// TwinCAT 3 PLC project CarlPlc
// ProgramVersion: 3.1.4022.1
// libraries:
//   Tc2_ModbusRTU, * (Beckhoff Automation GmbH)
//   Tc2_Standard, * (Beckhoff Automation GmbH)
//   Tc2_System, * (Beckhoff Automation GmbH)
//   Tc2_Utilities, * (Beckhoff Automation GmbH)
//   Tc3_Module, * (Beckhoff Automation GmbH)
//   BASIC,3.3.3.0,OSCAT
// project tree:
//   Common/ DetectEvent.TcPOU (not stored), GVL_Common.TcGVL (not stored), TasterEventStates.TcDUT, TasterEventType.TcDUT (not stored), LinearCalibration.TcDUT (not stored)
//   FlowRateSensor/ GVL_FlowControl.TcGVL (not stored), PRG_UpdateFlowRateSensor.TcPOU
//   GasAnalysis/ GVL_GasAnalysis.TcGVL, PRG_GasAnalysis.TcPOU (not stored)
//   GasSupply/ GVL_GasSupply.TcGVL (not stored), PRG_UpdateGasSupply.TcPOU (not stored)
//   MotorControl/ GVL_MotorControl.TcGVL, PRG_UpdateMotor.TcPOU (not stored)
//   pHOrpControl/ EN_ModbusReadTarget.TcDUT (not stored), GVL_PhOrpControl.TcGVL (not stored), PRG_ReadModbusSensorData.TcPOU, PRG_UpdatePhControl.TcPOU (not stored)
//   / PlcTask.TcTTO (not stored)
//   MAIN/ MAIN.TcPOU (not stored)
//   ReactorPressureControl/ GVL_ReactorPressureControl.TcGVL (not stored), PRG_UpdatePressureSensor.TcPOU (not stored)
//   RoomTempRh/ GVL_TempRHSensor.TcGVL, PRG_UpdateRoomTempRh.TcPOU (not stored)
//   TemperatureControl/ EN_TempControlMode.TcDUT (not stored), FB_TON.TcPOU (not stored), GVL_TemperatureControl.TcGVL, FUN_ComputeMovingSetPoint.TcPOU, PRG_UpdateTemperatureControl.TcPOU
//   TemperatureControl/PID/ CLK_PRG.TcPOU, FB_PWM.TcPOU (not stored), FT_DERIV.TcPOU (not stored), FT_PIDWL.TcPOU, FT_PIWL.TcPOU, PWM_DC.TcPOU (not stored), TP_X.TcPOU (not stored), T_PLC_MS.TcPOU (not stored), T_PLC_US.TcPOU
// real-time tasks:
//   TASK PlcTask: cycle T#10ms, priority 20, ADS port 350
// I/O:
//   DEVICE Device 1 (EtherCAT), AmsNetId 5.54.16.198.2.1
//     Term 1 (EK1200) [EK1200-5000 EtherCAT Power supply (2A E-Bus)]
//       Term 2 (EL3014) Motor Speed In [EL3014 4Ch. Ana. Input 0-20mA DIFF]
//       Term 3 (EL4004) Motor Speed Out [EL4004 4Ch. Ana. Output 0-10V, 12bit]
//       Term 4 (EL2004) DO Heating Cooling [EL2004 4Ch. Dig. Output 24V, 0.5A]
//       Term 5 (EL2004) DO Gassing Valves [EL2004 4Ch. Dig. Output 24V, 0.5A]
//       Term 6 (EL2004) DO Motor Control Out [EL2004 4Ch. Dig. Output 24V, 0.5A]
//       Term 7 (EL6021) PhModbus [EL6021 Interface (RS422/485)]
//       Term 8 (EL6021) OrpModbus [EL6021 Interface (RS422/485)]
//       Term 21 (EL1004) DI Gas Analysis [EL1004 4Ch. Dig. Input 24V, 3ms]
//       Term 18 (EL3052) AI Pressure Flow [EL3052 2Ch. Ana. Input 4-20mA]
//       Term 24 (EL3052) AI Heating Cooling [EL3052 2Ch. Ana. Input 4-20mA]
//       Term 10 (EL9184) [EL9184 Potential Connection, 8 x 24V, 8 x Ground]
//       Term 26 (EL3044) [EL3044 4Ch. Ana. Input 0-20mA]
//       Term 9 (EL9011) [EL9011 End Terminal]
// variable links:
//   CarlPlc/CarlPlc Instance <-> Device 1 (EtherCAT)/Term 1 (EK1200)/Term 18 (EL3052) AI Pressure Flow
//     PlcTask Inputs/GVL_FlowControl.flowRateRawCounts <-> FlowRateSensor/FlowRateRaw
//     PlcTask Inputs/GVL_ReactorPressureControl.pressureRawCounts <-> PressureSensor/PressureSensorRaw
//   CarlPlc/CarlPlc Instance <-> Device 1 (EtherCAT)/Term 1 (EK1200)/Term 2 (EL3014) Motor Speed In
//     PlcTask Inputs/GVL_MotorControl.motorActualSpeed <-> AI Motor RPM/Value
//     PlcTask Inputs/GVL_TempRHSensor.roomRhRaw <-> AI Room RH/Value
//     PlcTask Inputs/GVL_TempRHSensor.roomTempRaw <-> AI Room Temp/Value
//   CarlPlc/CarlPlc Instance <-> Device 1 (EtherCAT)/Term 1 (EK1200)/Term 21 (EL1004) DI Gas Analysis
//     PlcTask Inputs/GVL_GasAnalysis.ch4FlowSensor <-> Flow Sensor CH4/Input
//     PlcTask Inputs/GVL_GasAnalysis.o2FlowSensor <-> Flow Sensor O2/Input
//   CarlPlc/CarlPlc Instance <-> Device 1 (EtherCAT)/Term 1 (EK1200)/Term 24 (EL3052) AI Heating Cooling
//     PlcTask Inputs/GVL_TemperatureControl.jacketTempRaw <-> AI Jacket Temp/Value
//   CarlPlc/CarlPlc Instance <-> Device 1 (EtherCAT)/Term 1 (EK1200)/Term 26 (EL3044)
//     PlcTask Inputs/GVL_GasAnalysis.ch4SensorRaw <-> AI CH4/Value
//     PlcTask Inputs/GVL_GasAnalysis.o2SensorRaw <-> AI O2/Value
//     PlcTask Inputs/GVL_GasSupply.gasSupplyPressureRaw <-> AI Gas Supply Pressure/Value
//   CarlPlc/CarlPlc Instance <-> Device 1 (EtherCAT)/Term 1 (EK1200)/Term 3 (EL4004) Motor Speed Out
//     PlcTask Outputs/GVL_MotorControl.motorTargetSpeed <-> MotorTargetSpeed/MotorTargetSpeed
//     PlcTask Outputs/GVL_PhOrpControl.acidPumpSpeedCount <-> AcidPumpSpeedCount/acidPumpSpeedCount
//   CarlPlc/CarlPlc Instance <-> Device 1 (EtherCAT)/Term 1 (EK1200)/Term 4 (EL2004) DO Heating Cooling
//     PlcTask Outputs/GVL_TemperatureControl.coldValve <-> ColdValve/Output
//     PlcTask Outputs/GVL_TemperatureControl.hotValve <-> HotValve/Output
//     PlcTask Outputs/GVL_TemperatureControl.pumpOn <-> PumpOn/Output
//     PlcTask Outputs/GVL_TemperatureControl.steriValve <-> SteriValve/Output
//   CarlPlc/CarlPlc Instance <-> Device 1 (EtherCAT)/Term 1 (EK1200)/Term 5 (EL2004) DO Gassing Valves
//     PlcTask Outputs/GVL_GasSupply.gasSupplyValve <-> GasSupplyValve/Output
//     PlcTask Outputs/GVL_ReactorPressureControl.reactorPressureInletValve <-> reactorPressureInlet/ReactorPressureInlet
//     PlcTask Outputs/GVL_ReactorPressureControl.reactorPressureOutletValve <-> reactorPressureOutlet/Output
//   CarlPlc/CarlPlc Instance <-> Device 1 (EtherCAT)/Term 1 (EK1200)/Term 6 (EL2004) DO Motor Control Out
//     PlcTask Outputs/GVL_MotorControl.motorReset <-> motorReset/Output
//     PlcTask Outputs/GVL_MotorControl.motorStart <-> motorStart/Output
//   CarlPlc/CarlPlc Instance <-> Device 1 (EtherCAT)/Term 1 (EK1200)/Term 7 (EL6021) PhModbus
//     PlcTask Inputs/GVL_Common.PhModbus.InData/D[{0..21}] <-> COM TxPDO-Map Inputs/Data In {0..21}  (22 links)
//     PlcTask Inputs/GVL_Common.PhModbus.InData/Status <-> COM TxPDO-Map Inputs/Status
//     PlcTask Outputs/GVL_Common.PhModbus.OutData/Ctrl <-> COM RxPDO-Map Outputs/Ctrl
//     PlcTask Outputs/GVL_Common.PhModbus.OutData/D[{0..21}] <-> COM RxPDO-Map Outputs/Data Out {0..21}  (22 links)
//   CarlPlc/CarlPlc Instance <-> Device 1 (EtherCAT)/Term 1 (EK1200)/Term 8 (EL6021) OrpModbus
//     PlcTask Inputs/GVL_Common.OrpModbus.InData/D[{0..21}] <-> COM TxPDO-Map Inputs/Data In {0..21}  (22 links)
//     PlcTask Inputs/GVL_Common.OrpModbus.InData/Status <-> COM TxPDO-Map Inputs/Status
//     PlcTask Outputs/GVL_Common.OrpModbus.OutData/Ctrl <-> COM RxPDO-Map Outputs/Ctrl
//     PlcTask Outputs/GVL_Common.OrpModbus.OutData/D[{0..21}] <-> COM RxPDO-Map Outputs/Data Out {0..21}  (22 links)

// ---- Common/TasterEventStates.TcDUT
TYPE TasterEventStates : (TASTEVTST_Init := 0,
						TASTEVTST_FirstPosEdge,
						TASTEVTST_FirstNegEdge,
						TASTEVTST_FirstLongClick);
END_TYPE

// ---- GasAnalysis/GVL_GasAnalysis.TcGVL
VAR_GLOBAL
	ch4FlowSensor			AT %I*	: BOOL;
	o2FlowSensor			AT %I*	: BOOL;
	
	ch4SensorRaw			AT %I*	: INT;
	o2SensorRaw 			AT %I*	: INT;
	
	ch4ValuemA				: REAL := 0.0;
	o2ValuemA				: REAL := 0.0;
	
	ch4ValuePercent			: REAL := 0.0;
	o2ValuePercent			: REAL := 0.0;
	
	ch4CalibrationToPercent : LinearCalibration := (scaleFactor := 8.3415719228868017795353435491844E-5, offset := 0.3);
	ch4CalibrationToMa		: LinearCalibration := (scaleFactor := 20.0/32768.0, offset := 0.0);
	o2CalibrationToPercent	: LinearCalibration := (scaleFactor := 8.3415719228868017795353435491844E-5, offset := 0.3);
	o2CalibrationToMa		: LinearCalibration := (scaleFactor := 20.0/32768.0, offset := 0.0);
	
	(* Sensor Status *)
	ch4SensorStatus			: INT  := 0; 	(* 0: FAULT (1mA output), 1: BEAMBLOCK(2mA output), 2: STARTUP (3mA output), 3: Running (4 > 20 mA output) *)

	o2SensorFault			: BOOL := FALSE;
	
	gasAnalysisControlStartStop : BOOL := FALSE;
	gasAnalysisControlManual	: BOOL := FALSE;
	
	gasAnalysisValveAutomatic	: BOOL := FALSE;
	gasAnalysisValveManual 		: BOOL := FALSE;	

END_VAR


VAR_GLOBAL PERSISTENT
	ch4ValuePercentSet			: REAL := 0.0;
	gasAnalysisControlRunning 	: BOOL;
END_VAR

// ---- MotorControl/GVL_MotorControl.TcGVL
VAR_GLOBAL
	(* agitation motor *)	
	motorActualSpeed 	AT %I*	: INT;
	motorTargetSpeed 	AT %Q*	: INT;
	
	motorRpm					: INT; 
	
	(* motor target speed setting --> see retains *)
	motorStart			AT %Q*	: BOOL := FALSE;
	motorReset			AT %Q*	: BOOL := FALSE;
	
	motorStartButton			: BOOL := FALSE;
	motorStopButton				: BOOL := FALSE;
	motorResetButton			: BOOL := FALSE;

	(* motorIsRunning				: BOOL := FALSE; *)
END_VAR

VAR_GLOBAL PERSISTENT
	motorRunning				: BOOL;
	currentMotorSpeedSetting	: INT;
END_VAR

// ---- RoomTempRh/GVL_TempRHSensor.TcGVL
VAR_GLOBAL
	roomTempRaw			AT %I*	: INT;
	roomRhRaw 			AT %I*	: INT;	
	
	roomTemp			: REAL;
	roomRh				: REAL;
END_VAR

// ---- TemperatureControl/GVL_TemperatureControl.TcGVL
VAR_GLOBAL


	tPhCurrent					: REAL := 0.0;
	tPhLastReadingValid			: BOOL := FALSE;
	tOrpCurrent					: REAL := 0.0;
	tOrpLastReadingValid		: BOOL := FALSE;


	(* temperature control *)
	pumpOn				AT %Q* 	: BOOL := FALSE;
	coldValve			AT %Q* 	: BOOL := FALSE;
	hotValve			AT %Q* 	: BOOL := FALSE;
	steriValve			AT %Q*	: BOOL := FALSE; 
	
	jacketTempRaw		AT %I*	: INT;
	jacketTempC					: REAL := 0.0;
	jacketTempK					: REAL := 0.0;
	
	
	tempControlStop				: BOOL := FALSE;
	tempControlStart			: BOOL := FALSE;
	hotValveButton				: BOOL := FALSE;
	coldValveButton				: BOOL := FALSE;
	
	pumpIsRunning				: BOOL := FALSE;
	tempControlRunning			: BOOL := FALSE;
	tempSafetyEnabled			: BOOL := FALSE;
	
	steriStart					: BOOL := FALSE;
	steriStop					: BOOL := FALSE;
	steriRunning				: BOOL := FALSE;

	
	currentMeanTemp				: REAL := 0;
	currentTempValid			: BOOL := FALSE;
	(* target temp -> see retains *) 
	
	tempIsBelowSteriTemp		: BOOL := TRUE;
	(* target steri temp --> see retains *)	

	
END_VAR

VAR_GLOBAL PERSISTENT
	targetControlTemp			: REAL;
	targetSteriTemp				: REAL;
	targetSteriTimeMinutes		: INT;
	remainingSteriTimeMinutes	: REAL;
	
	
	remainingSteriTimeInMs		: DINT; (* 30 min in ms *)
	
	countTempSpikes				: INT;
	countValveMaxTimeExceeded	: INT;

	pidResetCounter				: INT;
END_VAR

VAR_GLOBAL CONSTANT
	CYCLE_TIME_IN_MS		: TIME := T#10ms;
END_VAR

// ---- pHOrpControl/PRG_ReadModbusSensorData.TcPOU
PROGRAM PRG_ReadModbusSensorData
VAR
	
	CurrentReadTarget			: EN_ModbusReadTarget := EN_ModbusReadTarget.READ_TARGET_PH;
	
	ProcessValueRegister		: WORD := 2089;
	TemperatureRegister			: WORD := 2409;
	PhSensorUnitId				: BYTE := 1;
	OrpSensorUnitId				: BYTE := 2;
	RegQuantityToRead			: WORD :=10;
	
	currentUnitId				: BYTE := PhSensorUnitId;
	currentModbusRegister		: WORD := ProcessValueRegister;

	ModbusBusy					: BOOL := FALSE;

	(* diagnostics *)	
	LastModbusError				: ST_ModbusErrorDiagnostics;
	LastErrorstate				: INT;
	CurrentState				: INT;
	CounterError				: INT := 0;
	CounterSuccess				: INT := 0;
	
	firstCall					: BOOL := TRUE;	
	
	scaleFactorPh				: REAL :=   1.219512195; (* 0.980167935 *);  		
	offsetPh					: REAL := 	-1.280487805; (* -0.0216290391086993 *);	


	scaleFactorOrp				: REAL := 0.999321727334388;
	offsetOrp					: REAL := 0.0;			
	
END_VAR

(* looping through pH, pH-T, ORP, ORP-T reading the latest values *)
IF firstCall THEN
	PhModbus.ReadRegs( Execute := FALSE);
	OrpModbus.ReadRegs( Execute := FALSE);
	firstCall := FALSE;
END_IF	

CASE  CurrentReadTarget OF 
	EN_ModbusReadTarget.READ_TARGET_PH:
		PhModbus.Readregs (UnitID 		:= PhSensorUnitId ,
   							Quantity   	:= RegQuantityToRead,
   							MBAddr    	:= ProcessValueRegister,
   							cbLength    := RegQuantityToRead*2,
   							pMemoryAddr := ADR(PhValueArrayIn),   
   							Execute    	:= TRUE,
   							Timeout    	:= T#300MS,
							Busy 		=> ModbusBusy	
						  );
		
		IF NOT ModbusBusy THEN
			PhModbus.ReadRegs(Execute:= FALSE);
			CurrentReadTarget := EN_ModbusReadTarget.READ_TARGET_PH_T;
	
			IF PhModbus.Error THEN
				LastModbusError 	:= PhModbus.ErrorDiagnostics;
				LastErrorstate 		:= CurrentState;
				CounterError 		:= CounterError + 1;
				phLastReadingValid 	:= FALSE;
			ELSE
				CounterSuccess 		:= CounterSuccess + 1;
				phLastReadingValid 	:= TRUE;
				phCurrent			:= PhValueArrayIn[1]*scaleFactorPh + offsetPh;
			END_IF
		END_IF
		
	EN_ModbusReadTarget.READ_TARGET_PH_T:
		PhModbus.Readregs (UnitID 		:= PhSensorUnitId ,
   							Quantity   	:= RegQuantityToRead,
   							MBAddr    	:= TemperatureRegister,
   							cbLength    := RegQuantityToRead*2,
   							pMemoryAddr := ADR(TPhValueArrayIn),   
   							Execute    	:= TRUE,
   							Timeout    	:= T#300MS,
							Busy 		=> ModbusBusy	
						  );
		
		IF NOT ModbusBusy THEN
			PhModbus.ReadRegs(Execute:= FALSE);	
			CurrentReadTarget := EN_ModbusReadTarget.READ_TARGET_ORP;

			IF PhModbus.Error THEN
				LastModbusError 	:= PhModbus.ErrorDiagnostics;
				LastErrorstate 		:= CurrentState;
				CounterError 		:= CounterError + 1;
				tPhLastReadingValid := FALSE;
			ELSE
				CounterSuccess 		:= CounterSuccess + 1;
				tPhLastReadingValid := TRUE;
				tPhCurrent			:= TPhValueArrayIn[1];
			END_IF
		END_IF
	
	EN_ModbusReadTarget.READ_TARGET_ORP:
		OrpModbus.Readregs (UnitID 		:= OrpSensorUnitId ,
   							Quantity   	:= RegQuantityToRead,
   							MBAddr    	:= ProcessValueRegister,
   							cbLength    := RegQuantityToRead*2,
   							pMemoryAddr := ADR(OrpValueArrayIn),   
   							Execute    	:= TRUE,
   							Timeout    	:= T#300MS,
							Busy 		=> ModbusBusy	
						  );
		
		IF NOT ModbusBusy THEN
			OrpModbus.ReadRegs(Execute:= FALSE);	
			CurrentReadTarget := EN_ModbusReadTarget.READ_TARGET_ORP_T;

			IF OrpModbus.Error THEN
				LastModbusError 	:= OrpModbus.ErrorDiagnostics;
				LastErrorstate 		:= CurrentState;
				CounterError 		:= CounterError + 1;
				orpLastReadingValid := FALSE;
			ELSE
				CounterSuccess 		:= CounterSuccess + 1;
				orpLastReadingValid := TRUE;
				orpCurrent			:= OrpValueArrayIn[1]*scaleFactorOrp + offsetOrp;
			END_IF
		END_IF

	EN_ModbusReadTarget.READ_TARGET_ORP_T:

		OrpModbus.Readregs (UnitID 		:= OrpSensorUnitId ,
   							Quantity   	:= RegQuantityToRead,
   							MBAddr    	:= TemperatureRegister,
   							cbLength    := RegQuantityToRead*2,
   							pMemoryAddr := ADR(TOrpValueArrayIn),   
   							Execute    	:= TRUE,
   							Timeout    	:= T#300MS,
							Busy 		=> ModbusBusy	
						  );
		
		IF NOT ModbusBusy THEN
			OrpModbus.ReadRegs(Execute:= FALSE);	
			CurrentReadTarget := EN_ModbusReadTarget.READ_TARGET_PH;

			IF OrpModbus.Error THEN
				LastModbusError := OrpModbus.ErrorDiagnostics;
				LastErrorstate 	:= CurrentState;
				CounterError 	:= CounterError + 1;
				tOrpLastReadingValid := FALSE;
			ELSE
				CounterSuccess 	:= CounterSuccess + 1;
				tOrpLastReadingValid := TRUE;
				tOrpCurrent	:= TOrpValueArrayIn[1];
			END_IF
		END_IF
	
END_CASE
			
IF tPhLastReadingValid AND tOrpLastReadingValid THEN
	currentMeanTemp := (tPhCurrent + tOrpCurrent)/2.0;
	currentTempValid := TRUE;
ELSIF tPhLastReadingValid AND NOT tOrpLastReadingValid THEN
	currentMeanTemp := tPhCurrent;
	currentTempValid := TRUE;
ELSIF NOT tPhLastReadingValid AND tOrpLastReadingValid THEN
	currentMeanTemp := tOrpCurrent;
	currentTempValid := TRUE;
ELSE 
	(* no valid temperature signal !! signal to stop temperature control, if active *)
	currentTempValid := FALSE;
END_IF

END_PROGRAM

// ---- FlowRateSensor/PRG_UpdateFlowRateSensor.TcPOU
PROGRAM PRG_UpdateFlowRateSensor
VAR
	deltaVolume : REAL := 0.0;
END_VAR

IF flowRateRawCounts < 20 THEN
	flowRateLitersPerMinute := 0.0;
ELSE
	flowRateLitersPerMinute := INT_TO_REAL(flowRateRawCounts)*flowRateCalibration.scaleFactor + flowRateCalibration.offset;
END_IF

deltaVolume := flowRateLitersPerMinute*0.01/60.0;
spargeVolume := spargeVolume + deltaVolume;
spargeVolumeCumulative := spargeVolumeCumulative+ deltaVolume;

IF  resetSpargeVolume THEN
	resetSpargeVolume := FALSE;
	spargeVolume := 0.0;
END_IF

IF resetSpargeVolumeCumulative THEN
	resetSpargeVolumeCumulative := FALSE;
	spargeVolumeCumulative := 0.0;
END_IF

END_PROGRAM

// ---- TemperatureControl/PID/CLK_PRG.TcPOU
	FUNCTION_BLOCK CLK_PRG
VAR_INPUT
	PT : TIME := t#10ms;
END_VAR
VAR_OUTPUT
	Q : BOOL;
END_VAR
VAR
	init : BOOL;
	last : TIME;
	tx: TIME;
END_VAR

(*clk_prg uses the internal sps time to generate a clock with programmable period time.
the period time is defined for 10ms .. 65s
the first cycle after start is a clk pulse and then depending on the programmed period time a delay.
every pulse is only valid for one cycle.
the accuracy of clk_prg is depending on the accuracy of the system clock.*)

(* read system time *)
tx := DWORD_TO_TIME(T_PLC_MS());

(* initialize on startup *)
IF NOT init THEN
	init := TRUE;
	last := tx - pt;
END_IF;

(* generate output pulse when next_pulse is reached *)
Q := tx - last >= pt;
IF Q THEN last := tx; END_IF;

END_FUNCTION_BLOCK

// ---- TemperatureControl/PID/FT_PIDWL.TcPOU
FUNCTION_BLOCK FT_PIDWL
VAR_INPUT
	IN : REAL;
	KP : REAL := 1.0;
	TN : REAL := 1.0;
	TV : REAL := 1.0;
	LIM_L : REAL := -1.0E38;
	LIM_H : REAL := 1.0E38;
	RST : BOOL;
END_VAR
VAR_OUTPUT
	Y : REAL;
	LIM : BOOL;
END_VAR
VAR
	piwl : FT_PIWL;
	diff : FT_DERIV;
END_VAR

(*
version 1.3	13. nov. 2009
programmer 	hugo
tested by		tobias

FT_PIDWL is a PID controller with dynamic wind_up reset.
The PID controller works according to the fomula Y = KP *(IN + KI * INTEG(e) + DERIV(e) ).
a rst will reset the integrator to 0
lim_h and Lim_l set the possible output range of the internal integrator.
the output flags lim will signal that the output limits are active.

default values for KP = 1, KI = 1, ILIM_L = -1E37, iLIM_H = +1E38.
*)

(* if rst then *)
IF rst THEN
	piwl(rst := TRUE);
	piwl.RST := FALSE;
ELSE
	(* run PIWL controller first *)
	(* we need to check if TN = 0 and do alternative calls *)
	IF TN = 0.0 THEN
		piwl(in := IN * KP, KP := 1.0, KI := 0.0, LIM_L := LIM_L, LIM_H := LIM_H);
	ELSE
		piwl(in := IN * KP, KP := 1.0, KI := 1.0 / TN, LIM_L := LIM_L, LIM_H := LIM_H);
	END_IF;

	(* run differentiator and add_to_output *)
	diff(IN := IN, K := TV);
	Y := piwl.Y + diff.out;

	(* limit the output *)
	IF Y < LIM_L THEN
		LIM := TRUE;
		Y := LIM_L;
	ELSIF Y > LIM_H THEN
		LIM := TRUE;
		Y := LIM_H;
	ELSE
		LIM := FALSE;
	END_IF;
END_IF;



(* revision history
hm 13. jun. 2008 	rev 1.0
	original version

hm	25. jan 2008	rev 1.1
	multiply differential part with KP

hm	11. mar. 2009	rev 1.2
	real constants updated to new systax using dot

hm	13. nov. 2009	rev 1.3
	fixed code for negative KP

*)

END_FUNCTION_BLOCK

// ---- TemperatureControl/PID/FT_PIWL.TcPOU
FUNCTION_BLOCK FT_PIWL
VAR_INPUT
	IN : REAL;
	KP : REAL ;
	KI : REAL ;
	LIM_L : REAL := -1.0E38;
	LIM_H : REAL := 1.0E38;
	RST : BOOL;
END_VAR
VAR_OUTPUT
	Y : REAL;
	LIM : BOOL;
END_VAR
VAR
	init: BOOL;
	tx: DWORD;
	tc : REAL;
	t_last: DWORD;
	in_last : REAL;
	i: REAL;
	p: REAL;
END_VAR

(*
version 1.3	11. mar. 2009
programmer 	hugo
tested by		oscat

FT_PIWL is a PI controller.
The PID controller works according to the fomula Y = IN *(KP+ KI * INTEG(e) ).
a rst will reset the integrator to 0
lim_h and Lim_l set the possible output range of the controller.
the output flag lim will signal that the output limits are active.
the integrator ist equipped with anti wind-up circuitry which limits trhe total output ranke to lim_l and lim_h

default values for KP = 1, KI = 1, ILIM_L = -1E37, iLIM_H = +1E38.
*)

(* initialize at power_up *)
IF NOT init OR RST THEN
	init := TRUE;
	in_last := in;
	t_last := T_PLC_US();
	i := 0.0;
	tc := 0.0;
ELSE
	(* read last cycle time in Microseconds *)
	tx := T_PLC_US();
	tc := DWORD_TO_REAL(tx - t_last);
	t_last := tx;

	(* calculate proportional part *)
	p := KP * IN;

	(* run integrator *)
	i := (IN + in_last) * KI * tc ;
	in_last := IN;

	(* calculate output Y *)
	Y := p + i;

	(* check output for limits *)
	IF Y >= LIM_H THEN
		Y := LIM_H;
		IF ki <> 0.0 THEN
			i := LIM_H - p;
		ELSE
			i := 0.0;
		END_IF;
		LIM := TRUE;
	ELSIF Y <= LIM_L THEN
		Y := LIM_L;
		IF ki <> 0.0 THEN
			i := LIM_L - p;
		ELSE
			i := 0.0;
		END_IF;
		LIM := TRUE;
	ELSE
		LIM := FALSE;
	END_IF;
END_IF;

END_FUNCTION_BLOCK

// ---- TemperatureControl/PID/T_PLC_US.TcPOU
FUNCTION T_PLC_US : DWORD
VAR CONSTANT
	debug : BOOL := 0;
	N : INT := 0;
	offset : DWORD := 0;
END_VAR
VAR
	tx : TIME;
END_VAR

(*
version 1.2	16 nov 2008
programmer 	hugo
tested by	tobias

T_PLC_US reads the internal PLC timer and return the time, it has the advantage to be able to set a debug mode 
and speed up the counter to test the plc timer overrun which occurs every 50 days respectively 25 days at siemens S7
this routine also allows to correct the behavior of s7 where the internal plc counter will not count all 32 bits.

*)

tx := TIME();
T_PLC_US := TIME_TO_DWORD(Tx)*1000;

IF debug THEN
	T_PLC_US := (SHL(T_PLC_US,N) OR SHL(DWORD#1,N)-1) + OFFSET;
END_IF;

(* revision history
hm	14.9.2007	rev 1.0
	original version

hm	12. nov 2007	rev 1.1
	added temporaray variable tx because some compilers could not handle time() as an argument

hm	16. nov. 2008	rev 1.2
	initialized constants with 0 for compatibility reasons

*)

END_FUNCTION

// ---- TemperatureControl/FUN_ComputeMovingSetPoint.TcPOU
FUNCTION FUN_ComputeMovingSetPoint : REAL
VAR_INPUT
	currentTemp 		: REAL;
	targetSetPoint 		: REAL;
END_VAR	
VAR
	deltaTemp 			: REAL;
	sign				: REAL;
	maxDeltaTemp		: REAL;
END_VAR

deltaTemp := targetSetPoint - currentTemp;
maxDeltaTemp := 10.0;

IF deltaTemp >= 0 THEN
	sign := 1.0;
ELSE
	sign := -1.0;
END_IF

IF ABS(deltaTemp) > maxDeltaTemp THEN
	FUN_ComputeMovingSetPoint := sign*maxDeltaTemp + currentTemp;
ELSE
	FUN_ComputeMovingSetPoint := targetSetPoint;
END_IF

END_FUNCTION

// ---- TemperatureControl/PRG_UpdateTemperatureControl.TcPOU
PROGRAM PRG_UpdateTemperatureControl
VAR
	tempControlMode				: EN_TempControlMode := EN_TempControlMode.TEMP_MODE_MANUAL;  
	
	loopCounter					: DINT := 0;

	(* Controller settings *)
	pwmPeriodinSec			: TIME := T#25S;
	pwmDutyCycle			: REAL := 0.0;	
	pwmOutputValveControl 	: FB_PWM;
	
	pidController			: FT_PIDWL;
	
	kp_heating				: REAL := 0.002;
	tv_heating				: REAL := 200;
	tn_heating				: REAL := 1800;
	
	kp_cooling				: REAL := 0.006;
	tv_cooling				: REAL := 200;
	tn_cooling				: REAL := 1800;

	kp_steri				: REAL := 0.0065;
	tv_steri				: REAL := 200;
	tn_steri				: REAL := 300;
	
	kp						: REAL := kp_heating;
	tv						: REAL := tv_heating;
	tn						: REAL := tn_heating;

	(* KD = KP*TV *)			
	(* KI = KP/TN *)
	
	errorTemp				: REAL := 0.0;
	pidReset				: BOOL := FALSE;
		
	evtSteriStart			: DetectEvent;
	evtSteriStop			: DetectEvent;
		
	evtTempControlStart		: DetectEvent;
	evtTempControlStop		: DetectEvent;
	
	windUpResetTimer		: TON;
	windUpResetTime			: TIME := T#30S;
	
	maxValveOnTimer		 	: TON;
	maxValveOnTime			: TIME := T#25S;	
	
	evtPidReset				: DetectEvent;
	(*
	myPwmBlock				: FB_PWM;
	pwmCycleTime			: TIME := T#2S;
	myPwmDutyCycle			: REAL := 0.5;
	*)
END_VAR

(* jacket temperature input *)
jacketTempC := INT_TO_REAL(jacketTempRaw)/32768.0*200.0 -50.0;
jacketTempK := jacketTempC + 273.15;
tOrpCurrent;

evtSteriStart(		newSignalValue := steriStart);
evtSteriStop(		newSignalValue := steriStop);
evtTempControlStart(newSignalValue := tempControlStart);
evtTempControlStop(	newSignalValue := tempControlStop);
evtPidReset( 		newSignalValue := pidReset);


IF evtSteriStart.eventDetected = TASTEVT_PositiveEdge THEN
	steriStart := FALSE;
	pumpOn := FALSE;
	pidController( RST:= TRUE );
	tempControlMode	:= EN_TempControlMode.TEMP_MODE_STERI;
	tempControlRunning := FALSE;
	steriRunning := TRUE;
	steriValve := FALSE;
	coldValve := FALSE;
	hotValve := FALSE;
	(* Set remaining steri temp *)
	remainingSteriTimeInMs := targetSteriTimeMinutes*60*1000; 
END_IF

IF evtTempControlStart.eventDetected = TASTEVT_PositiveEdge THEN
	tempControlStart := FALSE;
	pumpOn := FALSE;
	pidController( RST:= TRUE );
	tempControlMode	:= EN_TempControlMode.TEMP_MODE_HEATCOOL;
	tempControlRunning := TRUE;
	steriRunning := FALSE;
	steriValve := FALSE;
	coldValve := FALSE;
	hotValve := FALSE;
END_IF

IF 	evtSteriStop.eventDetected = TASTEVT_PositiveEdge OR
 	evtTempControlStop.eventDetected = TASTEVT_PositiveEdge 
THEN
	steriStop := FALSE;
	tempControlStop := FALSE;
	pumpOn := FALSE;
	pidController( RST:= TRUE );
	tempControlRunning := FALSE;
	steriRunning := FALSE;
	tempControlMode	:= EN_TempControlMode.TEMP_MODE_MANUAL;
	coldValve := FALSE;
	hotValve := FALSE;
	steriValve := FALSE;
	(* TODO: Reset Steri Timer *)
END_IF

CASE tempControlMode OF
	EN_TempControlMode.TEMP_MODE_MANUAL:
		pumpOn := FALSE;
		pidController( RST:= TRUE );
		
	EN_TempControlMode.TEMP_MODE_HEATCOOL:
	
		
		pumpOn := TRUE;
		(* errorTemp := targetControlTemp - currentMeanTemp; *)
		errorTemp := FUN_ComputeMovingSetPoint(currentTemp := currentMeanTemp, targetSetPoint := targetControlTemp) - currentMeanTemp;
		
		pidController(	IN:= errorTemp,
						KP:= kp,
						TN:= tn,
						TV:= tv,
						LIM_L:= -1.0,
						LIM_H:= 1.0,
						RST:= pidReset);
						
		(* pwmDutyCycle := ABS(pidController.Y); (* !! pwm block cannot handle negative inputs *) *)
		(* pwmDutyCycle := 0.05; *)
		
		
		pwmOutputValveControl(pwmCycleTime:=pwmPeriodinSec, pwmDutyCycle:=pwmDutyCycle);	
		
		
		IF pidController.Y > 0 THEN
			(* heating *)
			coldValve := FALSE;
			hotValve := pwmOutputValveControl.Q;
			kp := kp_heating;
			tv := tv_heating;
			tn := tn_heating;
			
		ELSE
			(* cooling *)
			coldValve := pwmOutputValveControl.Q;
			hotValve := FALSE;

			kp := kp_cooling;
			tv := tv_cooling;
			tn := tn_cooling;
		END_IF
		
	
	EN_TempControlMode.TEMP_MODE_STERI:
		pumpOn := FALSE;
		errorTemp := targetSteriTemp - currentMeanTemp;
		pidController(	IN:= errorTemp,
						KP:= kp_steri,
						TN:= tn_steri,
						TV:= tv_steri,
						LIM_L:= -1.0,
						LIM_H:= 1.0,
						RST:= pidReset);
						
		pwmDutyCycle := ABS(pidController.Y); (* !! pwm block cannot handle negative inputs *)
		
		pwmOutputValveControl(pwmCycleTime:=pwmPeriodinSec, pwmDutyCycle:=pwmDutyCycle);
				
		IF pidController.Y > 0 THEN
			(* heating *)
			coldValve := FALSE;
			steriValve := pwmOutputValveControl.Q;
		ELSE
			(* cooling *)
			(* coldValve := pwmOutputValveControl.Q; *)
			steriValve := FALSE;
		END_IF
		
		IF currentMeanTemp > (targetSteriTemp-0.5) THEN
			(* count down 10 ms each cycle *)
			remainingSteriTimeInMs := remainingSteriTimeInMs - 10;
			IF remainingSteriTimeInMs < 0 THEN
				tempControlMode := EN_TempControlMode.TEMP_MODE_MANUAL;
				steriValve := FALSE;
				coldValve := FALSE;
				steriStop := TRUE;
			END_IF
		END_IF		
		remainingSteriTimeMinutes := DINT_TO_REAL(remainingSteriTimeInMs)/(60.0*1000.0);
	
	
END_CASE

(*
maxValveOnTimer(IN:= (coldValve OR hotValve OR steriValve), PT:= maxValveOnTime);
IF maxValveOnTimer.Q THEN
	maxValveOnTimer(IN:=FALSE);
	countValveMaxTimeExceeded := countValveMaxTimeExceeded + 1;
	pidReset := TRUE;
	steriValve := FALSE;
	coldValve := FALSE;
	hotValve := FALSE;
END_IF
*)
(*
IF tempSafetyEnabled THEN
	IF (tPhLastReadingValid = FALSE AND tOrpLastReadingValid = FALSE) OR
		(currentMeanTemp > targetControlTemp + 0.5 OR currentMeanTemp < targetControlTemp - 0.5) THEN
		//tempControlMode := EN_TempControlMode.TEMP_MODE_MANUAL;
		pidReset := TRUE;
		countTempSpikes := countTempSpikes + 1;
		steriValve := FALSE;
		coldValve := FALSE;
		hotValve := FALSE;
	END_IF
END_IF
*)
 
IF evtPidReset.eventDetected = TASTEVT_PositiveEdge THEN
	pidReset := FALSE;
	pidController(RST:=TRUE);
	pidResetCounter := pidResetCounter + 1;
	steriValve := FALSE;
	coldValve := FALSE;
	hotValve := FALSE;
END_IF

END_PROGRAM
